{attribute 'linkalways'} 
{attribute 'no_explicit_call' := 'This FB is a CLASS and must be accessed using methods or properties'}
{attribute 'enable_dynamic_creation'}
FUNCTION_BLOCK FINAL ABS_INT EXTENDS Node
VAR
	in : _INT(0);
	out : _INT(0);
END_VAR

METHOD PUBLIC Clone : I_Node
VAR
	pNode : POINTER TO ABS_INT;
END_VAR
pNode := __NEW(ABS_INT);
Clone := pNode^;
END_METHOD

METHOD FB_init : BOOL
VAR_INPUT
	bInitRetains : BOOL; // if TRUE, the retain variables are initialized (warm start / cold start)
	bInCopyCode : BOOL;  // if TRUE, the instance afterwards gets moved into the copy code (online change)
END_VAR
AddInput('in',THIS^.in);
AddOutput('out', THIS^.out);
END_METHOD

METHOD PROTECTED OnExecute
VAR
END_VAR
out.Value := ABS(in.Value);
END_METHOD

END_FUNCTION_BLOCK

(* stored: Version 1.1.0.1, ProductVersion 3.1.4024.15
   POU ABS_INT: Id {96f4b1d4-719d-4ce3-a770-ecef2b91a911}, SpecialFunc None
   Folder Constructor: Id {230a924e-de2b-438e-ac09-220adaec4b73}
   Method Clone: Id {91dc8049-d92c-4e3f-b992-0c40e19faa97}
   Method FB_init: Id {4d820b9e-0ece-4cd4-992f-00eb1c823c8c}
   Method OnExecute: Id {28bc4da4-31f6-4a7b-a466-f8895a8316d9} *)
